(* CODESYS project MotorenInterface.project

Project tree, tasks and I/O mapping:
  CODESYS_Control_Win_V3 : CODESYS Control Win V3, 3S - Smart Software Solutions GmbH, version 3.5.13.20
    application Application
      task Task (cyclic, interval t#20ms, priority 1) calls Main
  interface MotorInterface: Start, Stop, Cycle, Initialize, MaxSpeed
  function block BenzineMotor [ST]: MaxSpeed, Start, Stop, Cycle, Initialize
  function block GasMotor [ST]: MaxSpeed, Start, Stop, Cycle, Initialize
  function block ElektroMotor [ST]: MaxSpeed, Start, Stop, Cycle, Initialize
  function block MotorBesturing [ST]: Start, Stop, Cycle, Initialize
  program Main [ST]
*)

// Main
PROGRAM Main
VAR
	fbMotorBesturing		: MotorBesturing;
END_VAR

END_PROGRAM

// MotorBesturing
FUNCTION_BLOCK MotorBesturing
VAR
	fbBenzineMotor		: BenzineMotor;			// Creëer Object van klasse BenzineMotor
	fbGasMotor			: GasMotor;				// Creëer Object van klasse GasMotor
	fbElektroMotor		: ElektroMotor;			// Creëer Object van klasse ElektroMotor
	iMotoren			: ARRAY [1..3] OF MotorInterface := [fbBenzineMotor, fbGasMotor, fbElektroMotor]; // Toekennen van de objecten aan de interface
END_VAR

METHOD Start
VAR
	i			: UINT;	
END_VAR
FOR i:= 1 TO 3 DO // Start alle motoren
	iMotoren[i].Start();
END_FOR;
END_METHOD

METHOD Stop
VAR
	i			: UINT;	
END_VAR
FOR i:= 1 TO 3 DO 
	iMotoren[i].Stop();
END_FOR;
END_METHOD

METHOD Cycle
VAR
	i			: UINT;
END_VAR
FOR i:= 1 TO 3 DO 
	iMotoren[i].Cycle();
END_FOR;
END_METHOD

METHOD Initialize
VAR
	
END_VAR
iMotoren[1].Initialize();
iMotoren[2].Initialize();
iMotoren[3].Initialize();
END_METHOD

END_FUNCTION_BLOCK

// BenzineMotor
FUNCTION_BLOCK BenzineMotor IMPLEMENTS MotorInterface
VAR
END_VAR

PROPERTY MaxSpeed : UINT
GET
END_GET
SET
END_SET
END_PROPERTY

METHOD Start
END_METHOD

METHOD Stop
END_METHOD

METHOD Cycle
END_METHOD

METHOD Initialize
END_METHOD

END_FUNCTION_BLOCK

// MotorInterface
INTERFACE MotorInterface

METHOD Start
VAR_INPUT
END_VAR
END_METHOD

METHOD Stop
VAR_INPUT
END_VAR
END_METHOD

METHOD Cycle
VAR_INPUT
END_VAR
END_METHOD

METHOD Initialize
VAR_INPUT
END_VAR
END_METHOD

PROPERTY MaxSpeed : UINT
SET
END_SET
GET
END_GET
END_PROPERTY

END_INTERFACE

// GasMotor
FUNCTION_BLOCK GasMotor IMPLEMENTS MotorInterface
VAR
END_VAR

PROPERTY MaxSpeed : UINT
GET
END_GET
SET
END_SET
END_PROPERTY

METHOD Start
END_METHOD

METHOD Stop
END_METHOD

METHOD Cycle
END_METHOD

METHOD Initialize
END_METHOD

END_FUNCTION_BLOCK

// ElektroMotor
FUNCTION_BLOCK ElektroMotor IMPLEMENTS MotorInterface
VAR
END_VAR

PROPERTY MaxSpeed : UINT
GET
END_GET
SET
END_SET
END_PROPERTY

METHOD Start
END_METHOD

METHOD Stop
END_METHOD

METHOD Cycle
END_METHOD

METHOD Initialize
END_METHOD

END_FUNCTION_BLOCK
